(* CoDeSys 2.3.9.50 project: Test.pro *)
(* Libraries: TcpIp.lib 31.8.18 23:12:47, TcBase.lib 14.5.09 11:14:08, TcSystem.lib 7.6.16 10:01:22, TcUtilities.lib 3.2.16 15:08:58, STANDARD.LIB 5.6.98 11:03:02, InfluxDB_1.0.0.0.lib 27.8.19 12:20:53, BinaryTool_1.0.0.0.lib 25.8.19 15:16:50 *)

(* Task configuration *)
TASK Standard (PRIORITY := 0, INTERVAL := T#10ms);
	MAIN();
END_TASK
TASK Writer (PRIORITY := 1, INTERVAL := T#10ms);
	Writer();
END_TASK

(* Global variable list: TwinCAT_Configuration *)
(* Generated automatically by TwinCAT - (read only) *)
VAR_CONFIG
	MAIN.EthernetDummy AT %IB0 : UINT;	(*  ~ {LinkedWith:TIID^Gerät 3 (RT-Ethernet)^Eingänge^DevState} *)
	MAIN.LizenzDummy AT %IB2 : UINT;	(*  ~ {LinkedWith:TIID^Gerät 1 (EtherCAT)^Klemme 1 (EK1200)^Klemme 2 (EL6070-1911)^InfoData^State} *)
	MAIN.Dummy AT %IB4 : UINT;	(*  ~ {LinkedWith:TIID^Gerät 1 (EtherCAT)^Eingänge^Frm0State} *)
END_VAR

(* POU MAIN, ST *)
PROGRAM MAIN
VAR
	(* MAIN variables *)

	fbRand				: DRAND;

	fbInfluxDB : FB_InfluxDB;
	rTest1 : REAL :=123.56;
	rTest2 : REAL :=124.56;
	rTest3 : REAL :=126.56;
	fbInfluxDB_StoreData : FB_InfluxDB_StoreData;
	fbR_TRIG 			: R_TRIG;
	fbTON				:TON := (PT := T#1m);
	fbTON2				:TON := (PT := T#90s);
END_VAR
fbTON(IN := TRUE);
fbTON2(IN := TRUE);

IF (fbTON.Q) THEN
	fbTON(IN := FALSE);
	fbRand();
	rTest1	:= LREAL_TO_REAL(fbRand.Num)*10;
	fbRand();
	rTest2	:= LREAL_TO_REAL(fbRand.Num)*15;
	fbRand();
	rTest3	:= LREAL_TO_REAL(fbRand.Num)*20;

	fbInfluxDB_StoreData(	i_sMeasurement	:= 'Testmeasurement',
						i_sSource		:= 'Testsource',
						i_sNameArg1  	:= 'MW_Real1',
						i_stArg1    		:= F_REAL (rTest1),
						i_sFormatArg1	:= '%.2f',
						i_sNameArg2  	:= 'MW_Real2',
						i_stArg2    		:= F_REAL (rTest2),
						i_sFormatArg2	:= '%.2f',
						i_sNameArg3  	:= 'MW_Real3',
						i_stArg3    		:= F_REAL (rTest3),
						i_sFormatArg3	:= '%.2f',
						io_fbInfluxDB_Fifo:= Writer.fbInfluxDB_Fifo
				 );

END_IF

IF (fbTON2.Q) THEN
	fbTON2(IN := FALSE);
	fbRand();
	rTest1	:= LREAL_TO_REAL(fbRand.Num)*10;
	fbRand();
	rTest2	:= LREAL_TO_REAL(fbRand.Num)*15;
	fbRand();
	rTest3	:= LREAL_TO_REAL(fbRand.Num)*20;

	fbInfluxDB_StoreData(	i_sMeasurement	:= 'Testmeasurement',
						i_sSource		:= 'Testsource2',
						i_sNameArg1  	:= 'MW_Real1',
						i_stArg1    		:= F_REAL (rTest1),
						i_sFormatArg1	:= '%.2f',
						i_sNameArg2  	:= 'MW_Real2',
						i_stArg2    		:= F_REAL (rTest2),
						i_sFormatArg2	:= '%.2f',
						i_sNameArg3  	:= 'MW_Real3',
						i_stArg3    		:= F_REAL (rTest3),
						i_sFormatArg3	:= '%.2f',
						io_fbInfluxDB_Fifo:= Writer.fbInfluxDB_Fifo
				 );

END_IF
END_PROGRAM

(* POU Writer, ST *)
PROGRAM Writer
VAR
	stInfluxDB_ConPar		: ST_InfluxDB_ConPar := (sIpv4Address:='',uPort:=8083,sHostName:='localhost',sDatabase:='db_measurements',sUser:='',sPassword:='');

	fbInfluxDB_Fifo		: FB_InfluxDB_Fifo;
	fbInfluxDB 			: FB_InfluxDB;
	fbR_TRIG 			: R_TRIG;

END_VAR
fbInfluxDB(io_stInfluxDB_ConPar:= stInfluxDB_ConPar, io_fbInfluxDB_Fifo:= fbInfluxDB_Fifo);

fbR_TRIG(CLK := fbInfluxDB.o_bError);
IF fbR_TRIG.Q THEN
	ADSLOGSTR(msgCtrlMask := ADSLOG_MSGTYPE_ERROR OR ADSLOG_MSGTYPE_LOG OR ADSLOG_MSGTYPE_STRING, msgFmtStr := 'Fehler :%s', strArg:=fbInfluxDB.o_sError);
END_IF
END_PROGRAM
